{library PUBLIC}
(*
Structure to handle datagrams on level 4.
*)
TYPE DataGram :
STRUCT
	ParameterDW:		DWORD;		(* Parameter value (32 bit), purpose dependent on type of function *)
	ParameterB:			BYTE;		(* Parameter value (8 bit), purpose dependent on type of function *)

	FunctionType:		BYTE;		(* Type of function (8 bit) specifies a set of functions, the number must be based on the enumeration FUNCTION_TYPE, note that an enumeration is 16 bit and must be converted with WORD_TO_BYTE() to fit in this structure *)
	FunctionNumber: 	BYTE;		(* Specific Function (8 bit) *)

	CheckSum:			BYTE;		(* Checksum for DataGram *)
END_STRUCT
END_TYPE

(* stored: Version 1.1.0.1, ProductVersion 3.1.4024.2
   DUT DataGram: Id {8eff609c-1264-4964-aa9f-498671fcd355} *)
